KUKA KRL program: chk_w3_grp1_clo.src

&ACCESS RVO1
&REL 2
&COMMENT Check GRP Z1 ACTROS CLOSE
DEF chk_w3_grp1_clo( )

; Check gripper actros CLOSE Z1.1 Z1.2
;//---- Start User-------

$TIMER[10] = 0
$TIMER_STOP[10] = FALSE

WAIT FOR ($IN[6] AND $IN[8])
WAIT FOR (NOT $IN[5] AND NOT $IN[7])

$TIMER_STOP[10] = TRUE
$TIMER[10] = 0

;//---- End User---------

END
